// TIA Portal V19 export
TYPE "_ILO_VM_Burkett8691rev3"
   STRUCT
      StandardStructure : Struct   // Burkett 8691 rev.2 DeviceID:
         Header : Struct
            NumberParameter : Int := 5;   // Number of device parameters (Device Identification + Device Parameter)
            AdressParamDownLoad : Int := 20;   // Start adress for ParamDownload signals in this struct
            AdressDeviceIndent : Int;   // Start adress for Device Identification Parameters in this struct (82 Bytes ea)
            AdressApplicSpez : Int;   // Start adress ApplicationSpezificTag (82 Bytes ea) [9]
            AdressDeviceParam : Int := 44;   // Start adress for Device Parameters in this Area (20 Bytes ea) [15]
            AdressKommando : Int;   // Start adress for Device Commandos
            NumberCommandos : Int;   // Number of Commandos of the device
            Spare01 : Int;   // spare
            Spare02 : Int;   // spare
            Spare03 : Int;   // spare
         END_STRUCT;
         Paramdownload : Struct
            ParamDownLoadStart : Struct   // Parameter Download Start (Only if master and device are V1.1)
               BlockStat : DWord;   // function block status
               IOLStat : DWord;   // IO-Link Status
            END_STRUCT;
            ParamDownLoadEnd : Struct   // Parameter Download End (Only if master and device are V1.1)
               BlockStat : DWord;   // function block status
               IOLStat : DWord;   // IO-Link Status
            END_STRUCT;
            ParamDownLoadStore : Struct   // Parameter Download Store (Only if master and device are V1.1)
               BlockStat : DWord;   // function block status
               IOLStat : DWord;   // IO-Link Status
            END_STRUCT;
         END_STRUCT;
         Parameter : Struct   // Address Device Indent
            ValveCyclesProgress : Struct   // Resettable
               value : Real;   // Percentage of ValveCyclesInterval
            END_STRUCT;
            Index : Int := 11270;   // parameter index
            Subindex : Int := 3;   // parameter subindex
            Length : Int := 4;   // parameter length in BYTE for writing
            BlockStat : DWord;   // function block status
            IOLStat : DWord;   // IO-Link Status
            RelRead : Bool := TRUE;   // reading release
            RelWrite : Bool;   // writing release
         END_STRUCT;
         Parameter1 : Struct   // Address Device Indent
            ValveCyclesInterval : Struct   // Resettable
               value : DInt;
            END_STRUCT;
            Index : Int := 11270;   // parameter index
            Subindex : Int := 4;   // parameter subindex
            Length : Int := 4;   // parameter length in BYTE for writing
            BlockStat : DWord;   // function block status
            IOLStat : DWord;   // IO-Link Status
            RelRead : Bool := TRUE;   // reading release
            RelWrite : Bool;   // writing release
         END_STRUCT;
         Parameter2 : Struct   // Address Device Indent
            SV1_EnDuration : Struct   // Opening Time (CMD)
               value : DInt;   // milliseconds
            END_STRUCT;
            Index : Int := 11279;   // parameter index
            Subindex : Int := 1;   // parameter subindex
            Length : Int := 4;   // parameter length in BYTE for writing
            BlockStat : DWord;   // function block status
            IOLStat : DWord;   // IO-Link Status
            RelRead : Bool := TRUE;   // reading release
            RelWrite : Bool;   // writing release
         END_STRUCT;
         Parameter3 : Struct   // Address Device Indent
            SV1_DeEnDuration : Struct   // Closing Time (CMD)
               value : DInt;   // milliseconds
            END_STRUCT;
            Index : Int := 11279;   // parameter index
            Subindex : Int := 2;   // parameter subindex
            Length : Int := 4;   // parameter length in BYTE for writing
            BlockStat : DWord;   // function block status
            IOLStat : DWord;   // IO-Link Status
            RelRead : Bool := TRUE;   // reading release
            RelWrite : Bool;   // writing release
         END_STRUCT;
         Parameter4 : Struct   // Address Device Indent
            ObjErrorTime : Struct
               value : DInt;   // Seconds
            END_STRUCT;
            Index : Int := 11279;   // parameter index
            Subindex : Int := 11;   // parameter subindex
            Length : Int := 4;   // parameter length in BYTE for writing
            BlockStat : DWord;   // function block status
            IOLStat : DWord;   // IO-Link Status
            RelRead : Bool := TRUE;   // reading release
            RelWrite : Bool;   // writing release
         END_STRUCT;
      END_STRUCT;
   END_STRUCT;
END_TYPE
